// Mitsubishi GX Works2 project: STEP_SEQUENCE   PLC: Q02/Q02H

PROGRAM MAIN
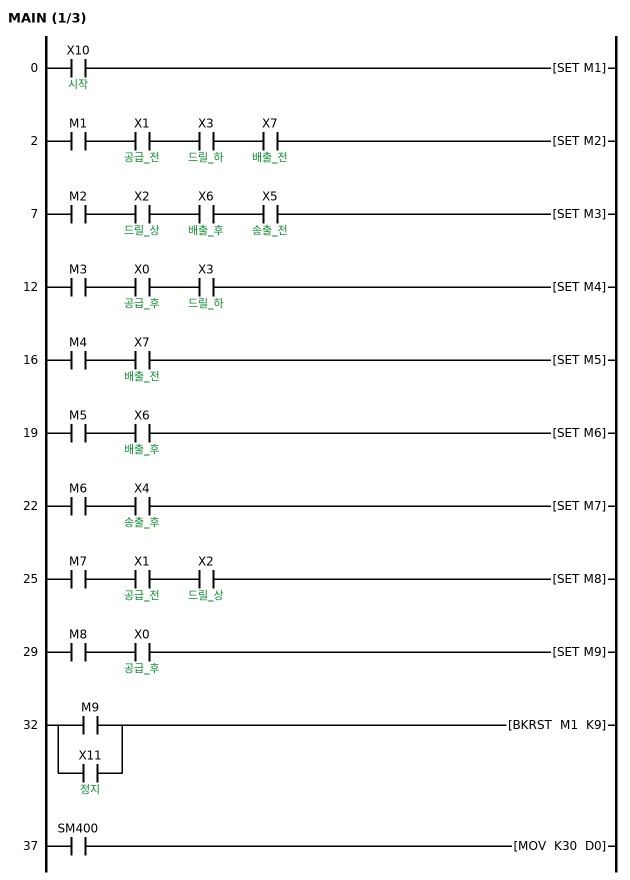
0     LD      X10  ; 시작
      SET     M1
2     LD      M1
      AND     X1  ; 공급_전
      AND     X3  ; 드릴_하
      AND     X7  ; 배출_전
      SET     M2
7     LD      M2
      AND     X2  ; 드릴_상
      AND     X6  ; 배출_후
      AND     X5  ; 송출_전
      SET     M3
12    LD      M3
      AND     X0  ; 공급_후
      AND     X3  ; 드릴_하
      SET     M4
16    LD      M4
      AND     X7  ; 배출_전
      SET     M5
19    LD      M5
      AND     X6  ; 배출_후
      SET     M6
22    LD      M6
      AND     X4  ; 송출_후
      SET     M7
25    LD      M7
      AND     X1  ; 공급_전
      AND     X2  ; 드릴_상
      SET     M8
29    LD      M8
      AND     X0  ; 공급_후
      SET     M9
32    LD      M9
      OR      X11  ; 정지
      BKRST   M1 K9
37    LD      SM400
      MOV     K30 D0
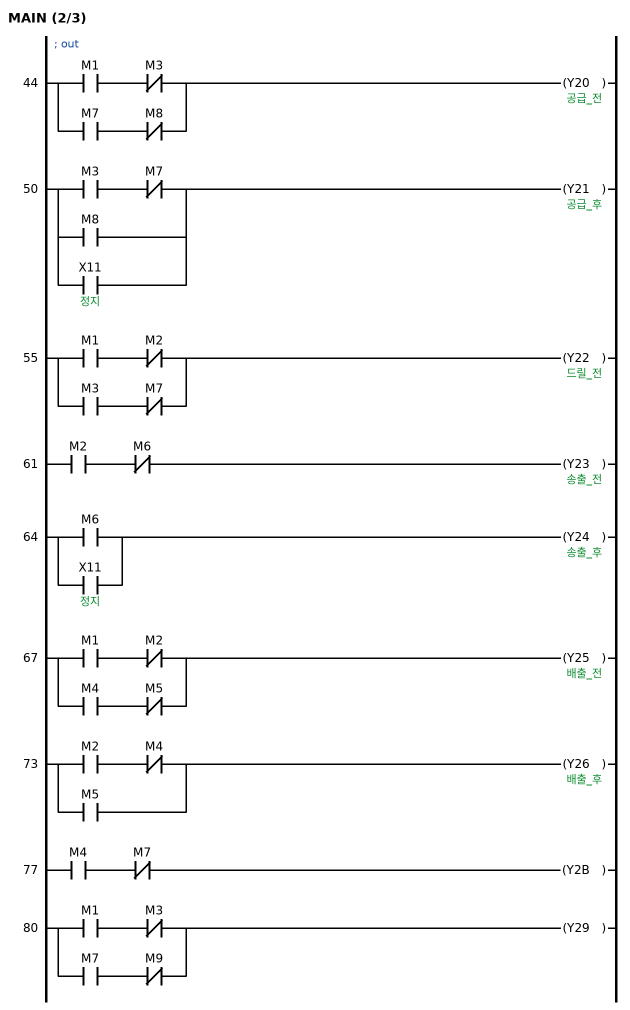
; out
44    LD      M1
      ANI     M3
      LD      M7
      ANI     M8
      ORB
      OUT     Y20  ; 공급_전
50    LD      M3
      ANI     M7
      OR      M8
      OR      X11  ; 정지
      OUT     Y21  ; 공급_후
55    LD      M1
      ANI     M2
      LD      M3
      ANI     M7
      ORB
      OUT     Y22  ; 드릴_전
61    LD      M2
      ANI     M6
      OUT     Y23  ; 송출_전
64    LD      M6
      OR      X11  ; 정지
      OUT     Y24  ; 송출_후
67    LD      M1
      ANI     M2
      LD      M4
      ANI     M5
      ORB
      OUT     Y25  ; 배출_전
73    LD      M2
      ANI     M4
      OR      M5
      OUT     Y26  ; 배출_후
77    LD      M4
      ANI     M7
      OUT     Y2B
80    LD      M1
      ANI     M3
      LD      M7
      ANI     M9
      ORB
      OUT     Y29
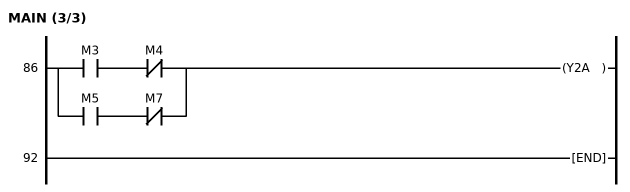
86    LD      M3
      ANI     M4
      LD      M5
      ANI     M7
      ORB
      OUT     Y2A
92    END
END_PROGRAM

PROGRAM APP1
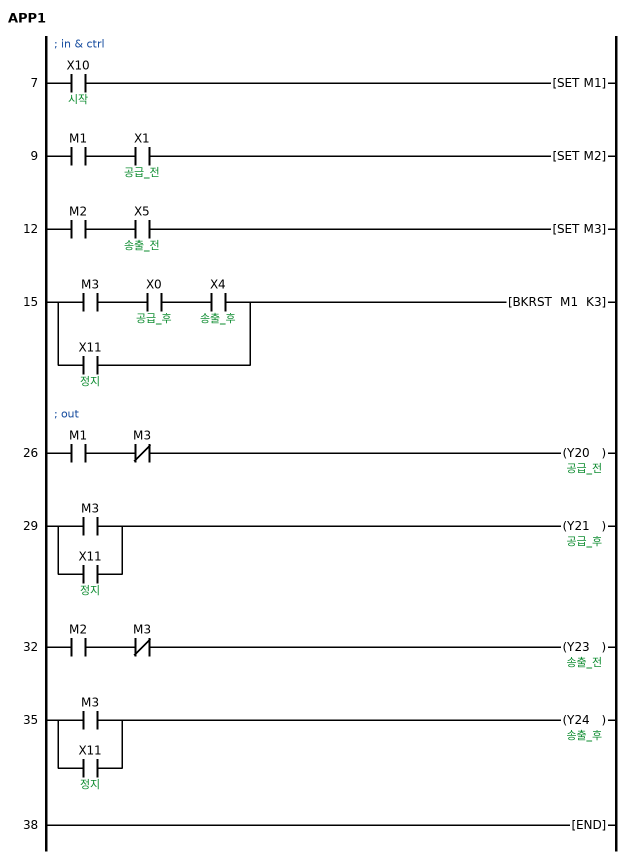
; in & ctrl
7     LD      X10  ; 시작
      SET     M1
9     LD      M1
      AND     X1  ; 공급_전
      SET     M2
12    LD      M2
      AND     X5  ; 송출_전
      SET     M3
15    LD      M3
      AND     X0  ; 공급_후
      AND     X4  ; 송출_후
      OR      X11  ; 정지
      BKRST   M1 K3
; out
26    LD      M1
      ANI     M3
      OUT     Y20  ; 공급_전
29    LD      M3
      OR      X11  ; 정지
      OUT     Y21  ; 공급_후
32    LD      M2
      ANI     M3
      OUT     Y23  ; 송출_전
35    LD      M3
      OR      X11  ; 정지
      OUT     Y24  ; 송출_후
38    END
END_PROGRAM

PROGRAM APP2
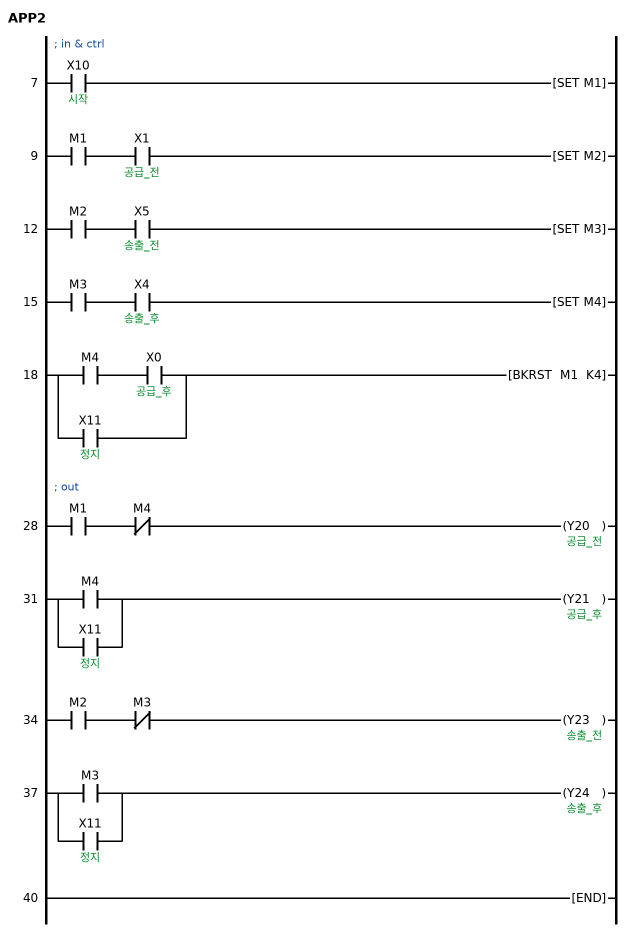
; in & ctrl
7     LD      X10  ; 시작
      SET     M1
9     LD      M1
      AND     X1  ; 공급_전
      SET     M2
12    LD      M2
      AND     X5  ; 송출_전
      SET     M3
15    LD      M3
      AND     X4  ; 송출_후
      SET     M4
18    LD      M4
      AND     X0  ; 공급_후
      OR      X11  ; 정지
      BKRST   M1 K4
; out
28    LD      M1
      ANI     M4
      OUT     Y20  ; 공급_전
31    LD      M4
      OR      X11  ; 정지
      OUT     Y21  ; 공급_후
34    LD      M2
      ANI     M3
      OUT     Y23  ; 송출_전
37    LD      M3
      OR      X11  ; 정지
      OUT     Y24  ; 송출_후
40    END
END_PROGRAM

PROGRAM APP3
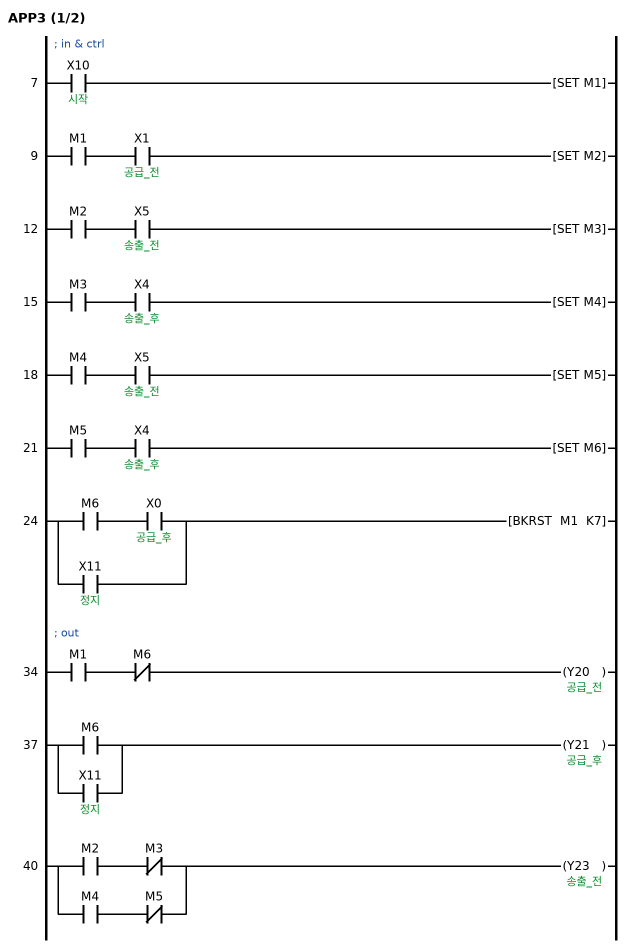
; in & ctrl
7     LD      X10  ; 시작
      SET     M1
9     LD      M1
      AND     X1  ; 공급_전
      SET     M2
12    LD      M2
      AND     X5  ; 송출_전
      SET     M3
15    LD      M3
      AND     X4  ; 송출_후
      SET     M4
18    LD      M4
      AND     X5  ; 송출_전
      SET     M5
21    LD      M5
      AND     X4  ; 송출_후
      SET     M6
24    LD      M6
      AND     X0  ; 공급_후
      OR      X11  ; 정지
      BKRST   M1 K7
; out
34    LD      M1
      ANI     M6
      OUT     Y20  ; 공급_전
37    LD      M6
      OR      X11  ; 정지
      OUT     Y21  ; 공급_후
40    LD      M2
      ANI     M3
      LD      M4
      ANI     M5
      ORB
      OUT     Y23  ; 송출_전
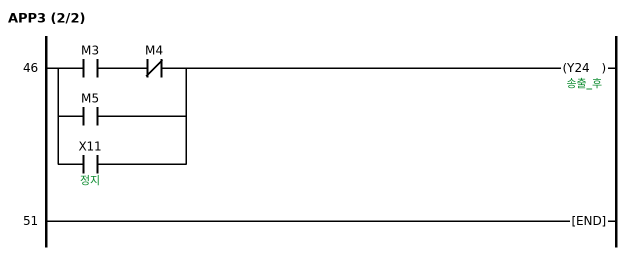
46    LD      M3
      ANI     M4
      OR      M5
      OR      X11  ; 정지
      OUT     Y24  ; 송출_후
51    END
END_PROGRAM

PROGRAM stepDoc
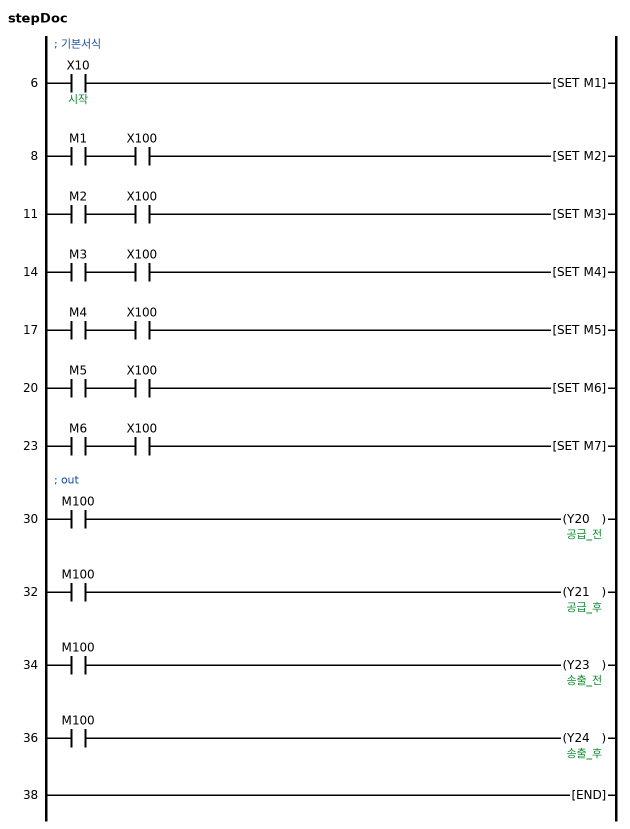
; 기본서식
6     LD      X10  ; 시작
      SET     M1
8     LD      M1
      AND     X100
      SET     M2
11    LD      M2
      AND     X100
      SET     M3
14    LD      M3
      AND     X100
      SET     M4
17    LD      M4
      AND     X100
      SET     M5
20    LD      M5
      AND     X100
      SET     M6
23    LD      M6
      AND     X100
      SET     M7
; out
30    LD      M100
      OUT     Y20  ; 공급_전
32    LD      M100
      OUT     Y21  ; 공급_후
34    LD      M100
      OUT     Y23  ; 송출_전
36    LD      M100
      OUT     Y24  ; 송출_후
38    END
END_PROGRAM

PROGRAM APP4
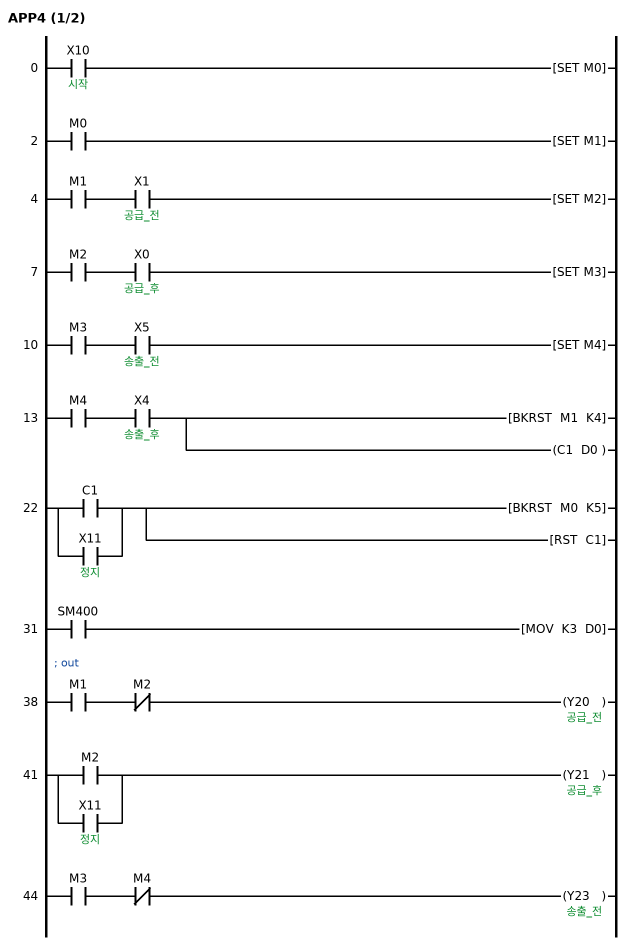
0     LD      X10  ; 시작
      SET     M0
2     LD      M0
      SET     M1
4     LD      M1
      AND     X1  ; 공급_전
      SET     M2
7     LD      M2
      AND     X0  ; 공급_후
      SET     M3
10    LD      M3
      AND     X5  ; 송출_전
      SET     M4
13    LD      M4
      AND     X4  ; 송출_후
      BKRST   M1 K4
      OUT     C1 D0
22    LD      C1
      OR      X11  ; 정지
      BKRST   M0 K5
      RST     C1
31    LD      SM400
      MOV     K3 D0
; out
38    LD      M1
      ANI     M2
      OUT     Y20  ; 공급_전
41    LD      M2
      OR      X11  ; 정지
      OUT     Y21  ; 공급_후
44    LD      M3
      ANI     M4
      OUT     Y23  ; 송출_전
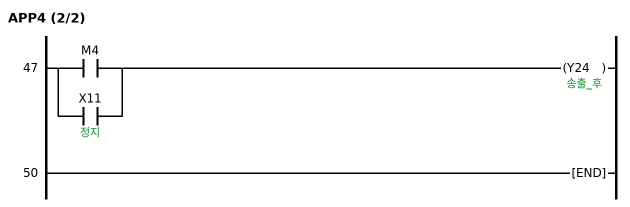
47    LD      M4
      OR      X11  ; 정지
      OUT     Y24  ; 송출_후
50    END
END_PROGRAM

PROGRAM APP3-1
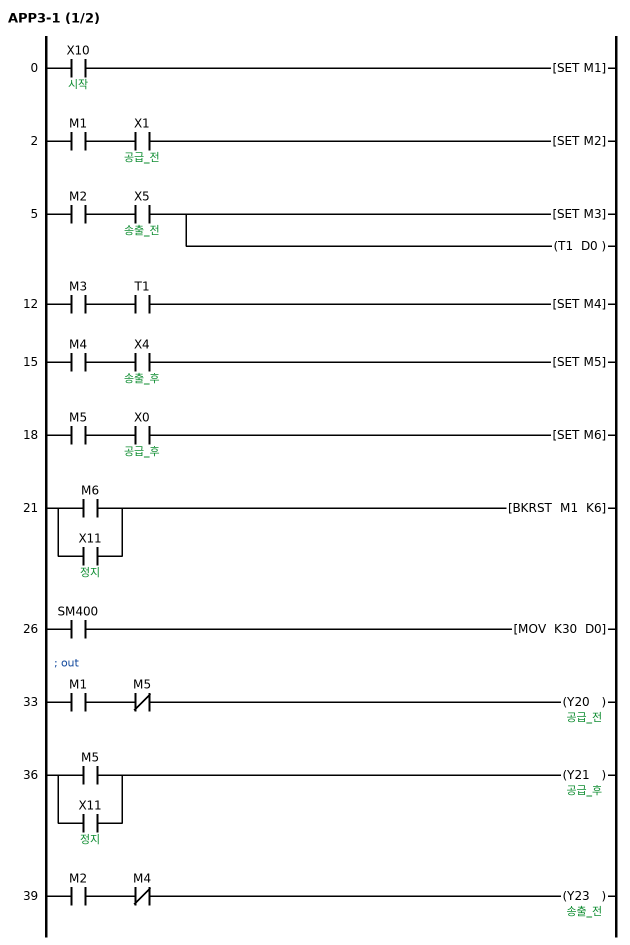
0     LD      X10  ; 시작
      SET     M1
2     LD      M1
      AND     X1  ; 공급_전
      SET     M2
5     LD      M2
      AND     X5  ; 송출_전
      SET     M3
      OUT     T1 D0
12    LD      M3
      AND     T1
      SET     M4
15    LD      M4
      AND     X4  ; 송출_후
      SET     M5
18    LD      M5
      AND     X0  ; 공급_후
      SET     M6
21    LD      M6
      OR      X11  ; 정지
      BKRST   M1 K6
26    LD      SM400
      MOV     K30 D0
; out
33    LD      M1
      ANI     M5
      OUT     Y20  ; 공급_전
36    LD      M5
      OR      X11  ; 정지
      OUT     Y21  ; 공급_후
39    LD      M2
      ANI     M4
      OUT     Y23  ; 송출_전
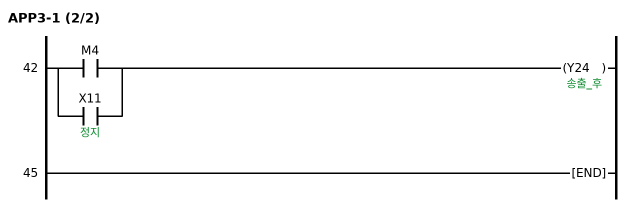
42    LD      M4
      OR      X11  ; 정지
      OUT     Y24  ; 송출_후
45    END
END_PROGRAM

PROGRAM complex1
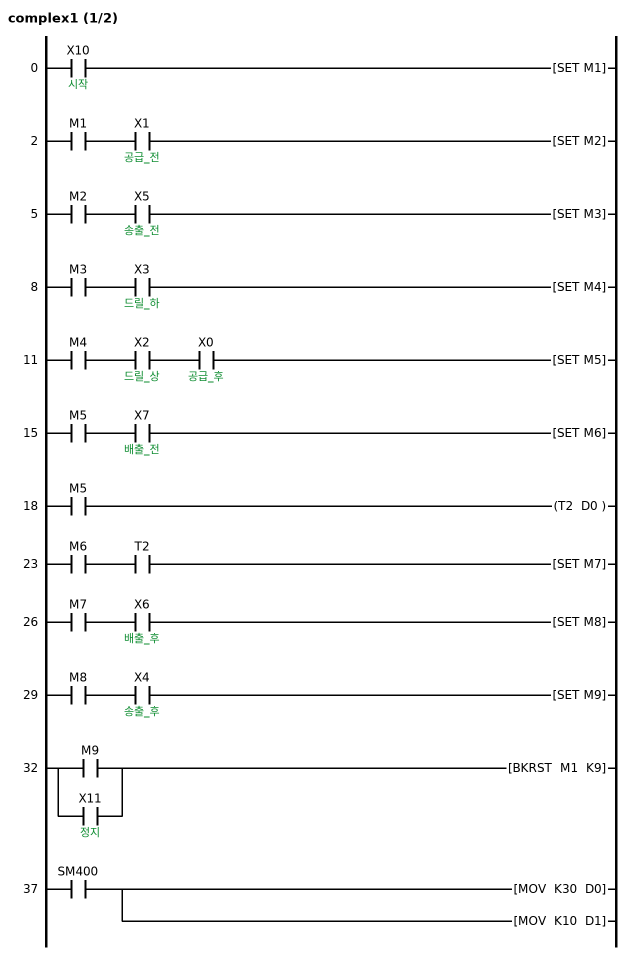
0     LD      X10  ; 시작
      SET     M1
2     LD      M1
      AND     X1  ; 공급_전
      SET     M2
5     LD      M2
      AND     X5  ; 송출_전
      SET     M3
8     LD      M3
      AND     X3  ; 드릴_하
      SET     M4
11    LD      M4
      AND     X2  ; 드릴_상
      AND     X0  ; 공급_후
      SET     M5
15    LD      M5
      AND     X7  ; 배출_전
      SET     M6
18    LD      M5
      OUT     T2 D0
23    LD      M6
      AND     T2
      SET     M7
26    LD      M7
      AND     X6  ; 배출_후
      SET     M8
29    LD      M8
      AND     X4  ; 송출_후
      SET     M9
32    LD      M9
      OR      X11  ; 정지
      BKRST   M1 K9
37    LD      SM400
      MOV     K30 D0
      MOV     K10 D1
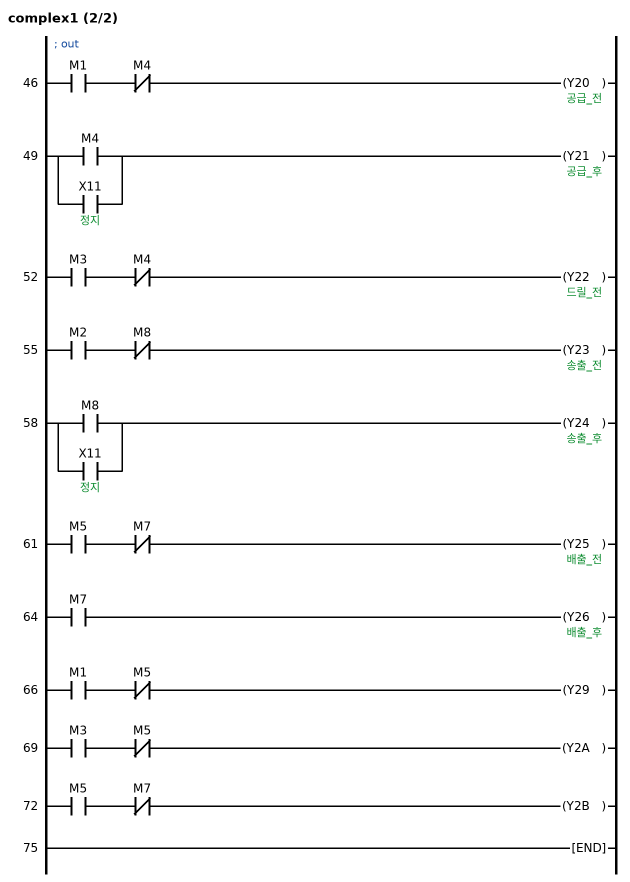
; out
46    LD      M1
      ANI     M4
      OUT     Y20  ; 공급_전
49    LD      M4
      OR      X11  ; 정지
      OUT     Y21  ; 공급_후
52    LD      M3
      ANI     M4
      OUT     Y22  ; 드릴_전
55    LD      M2
      ANI     M8
      OUT     Y23  ; 송출_전
58    LD      M8
      OR      X11  ; 정지
      OUT     Y24  ; 송출_후
61    LD      M5
      ANI     M7
      OUT     Y25  ; 배출_전
64    LD      M7
      OUT     Y26  ; 배출_후
66    LD      M1
      ANI     M5
      OUT     Y29
69    LD      M3
      ANI     M5
      OUT     Y2A
72    LD      M5
      ANI     M7
      OUT     Y2B
75    END
END_PROGRAM

PROGRAM complex2
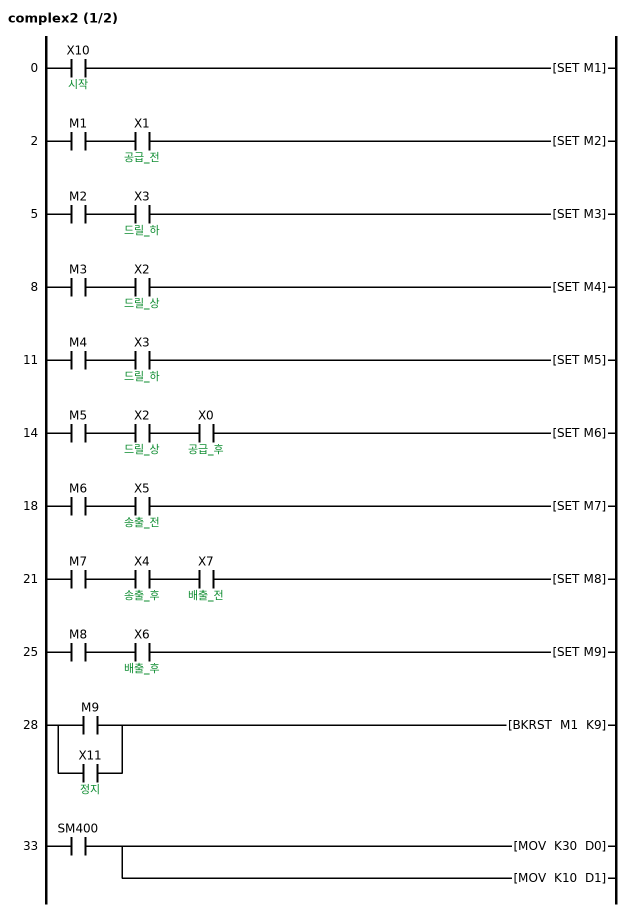
0     LD      X10  ; 시작
      SET     M1
2     LD      M1
      AND     X1  ; 공급_전
      SET     M2
5     LD      M2
      AND     X3  ; 드릴_하
      SET     M3
8     LD      M3
      AND     X2  ; 드릴_상
      SET     M4
11    LD      M4
      AND     X3  ; 드릴_하
      SET     M5
14    LD      M5
      AND     X2  ; 드릴_상
      AND     X0  ; 공급_후
      SET     M6
18    LD      M6
      AND     X5  ; 송출_전
      SET     M7
21    LD      M7
      AND     X4  ; 송출_후
      AND     X7  ; 배출_전
      SET     M8
25    LD      M8
      AND     X6  ; 배출_후
      SET     M9
28    LD      M9
      OR      X11  ; 정지
      BKRST   M1 K9
33    LD      SM400
      MOV     K30 D0
      MOV     K10 D1
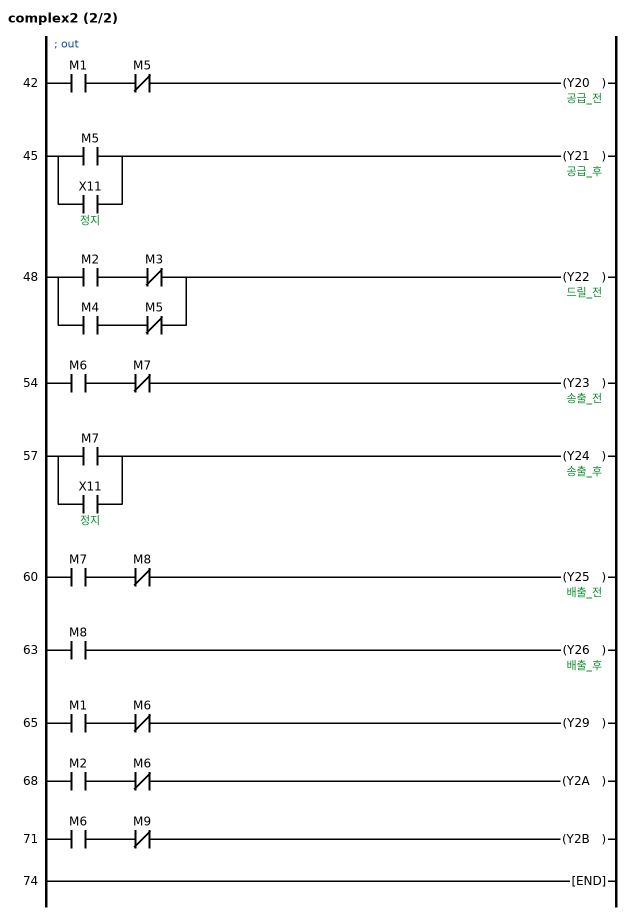
; out
42    LD      M1
      ANI     M5
      OUT     Y20  ; 공급_전
45    LD      M5
      OR      X11  ; 정지
      OUT     Y21  ; 공급_후
48    LD      M2
      ANI     M3
      LD      M4
      ANI     M5
      ORB
      OUT     Y22  ; 드릴_전
54    LD      M6
      ANI     M7
      OUT     Y23  ; 송출_전
57    LD      M7
      OR      X11  ; 정지
      OUT     Y24  ; 송출_후
60    LD      M7
      ANI     M8
      OUT     Y25  ; 배출_전
63    LD      M8
      OUT     Y26  ; 배출_후
65    LD      M1
      ANI     M6
      OUT     Y29
68    LD      M2
      ANI     M6
      OUT     Y2A
71    LD      M6
      ANI     M9
      OUT     Y2B
74    END
END_PROGRAM

PROGRAM complex3
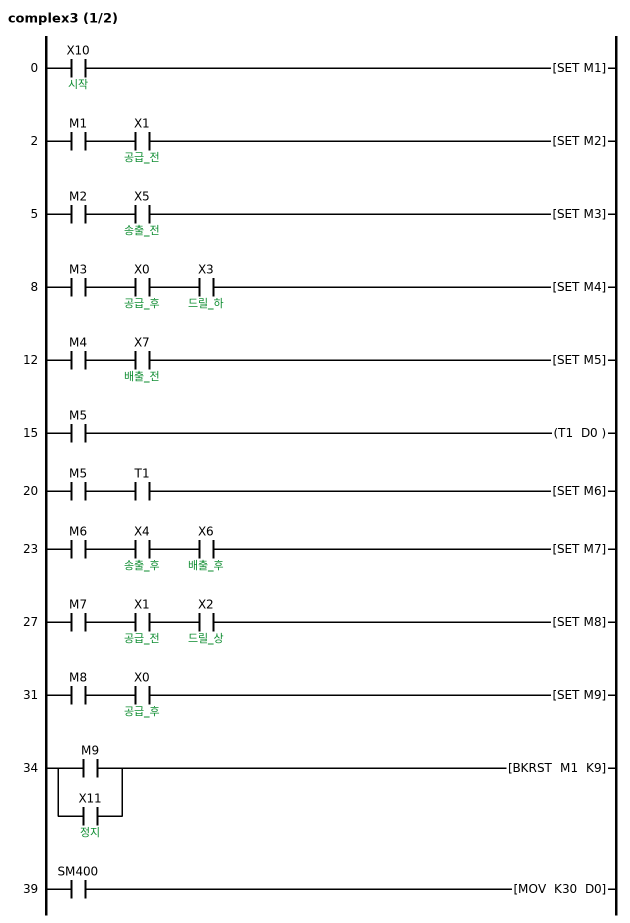
0     LD      X10  ; 시작
      SET     M1
2     LD      M1
      AND     X1  ; 공급_전
      SET     M2
5     LD      M2
      AND     X5  ; 송출_전
      SET     M3
8     LD      M3
      AND     X0  ; 공급_후
      AND     X3  ; 드릴_하
      SET     M4
12    LD      M4
      AND     X7  ; 배출_전
      SET     M5
15    LD      M5
      OUT     T1 D0
20    LD      M5
      AND     T1
      SET     M6
23    LD      M6
      AND     X4  ; 송출_후
      AND     X6  ; 배출_후
      SET     M7
27    LD      M7
      AND     X1  ; 공급_전
      AND     X2  ; 드릴_상
      SET     M8
31    LD      M8
      AND     X0  ; 공급_후
      SET     M9
34    LD      M9
      OR      X11  ; 정지
      BKRST   M1 K9
39    LD      SM400
      MOV     K30 D0
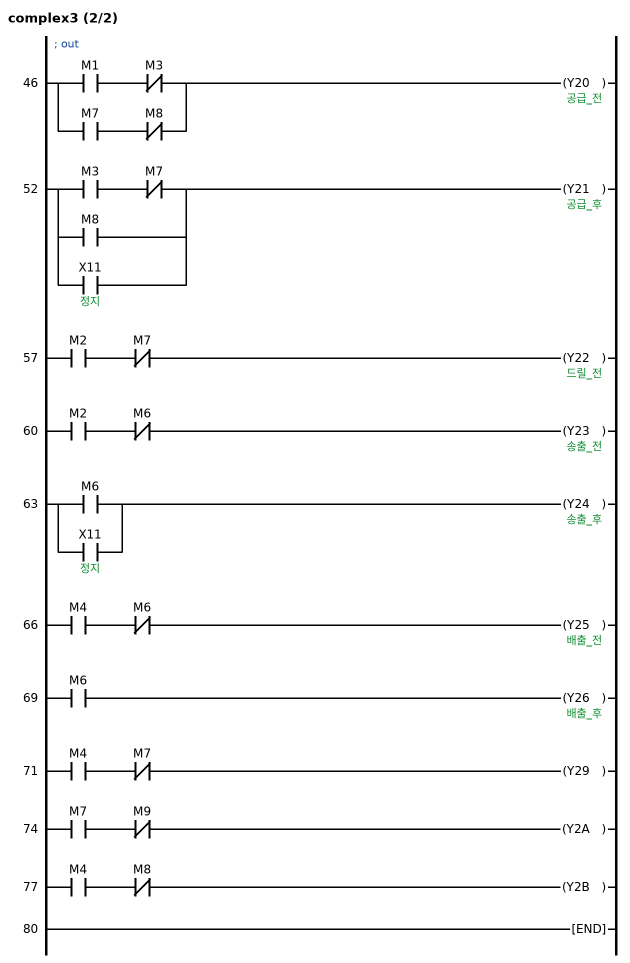
; out
46    LD      M1
      ANI     M3
      LD      M7
      ANI     M8
      ORB
      OUT     Y20  ; 공급_전
52    LD      M3
      ANI     M7
      OR      M8
      OR      X11  ; 정지
      OUT     Y21  ; 공급_후
57    LD      M2
      ANI     M7
      OUT     Y22  ; 드릴_전
60    LD      M2
      ANI     M6
      OUT     Y23  ; 송출_전
63    LD      M6
      OR      X11  ; 정지
      OUT     Y24  ; 송출_후
66    LD      M4
      ANI     M6
      OUT     Y25  ; 배출_전
69    LD      M6
      OUT     Y26  ; 배출_후
71    LD      M4
      ANI     M7
      OUT     Y29
74    LD      M7
      ANI     M9
      OUT     Y2A
77    LD      M4
      ANI     M8
      OUT     Y2B
80    END
END_PROGRAM

PROGRAM complex4
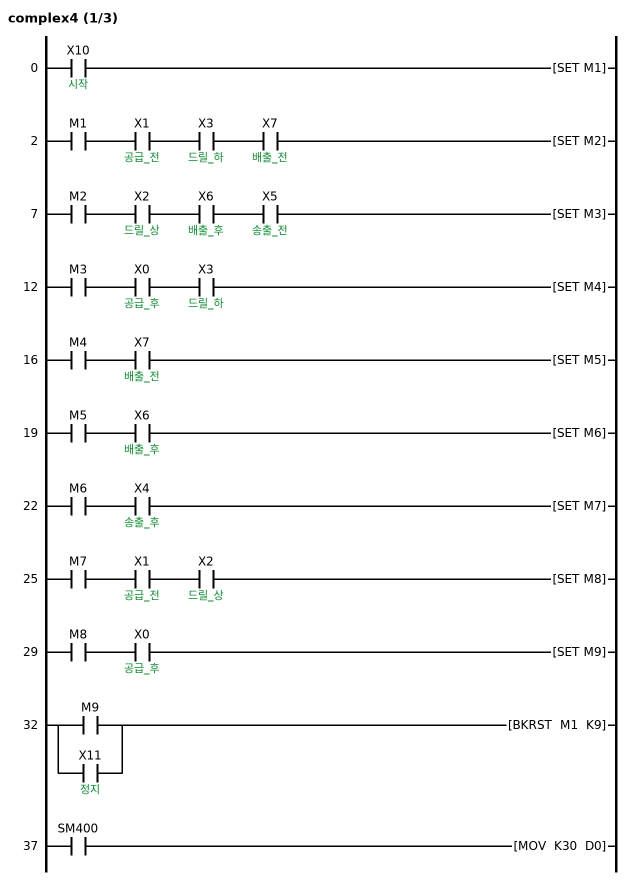
0     LD      X10  ; 시작
      SET     M1
2     LD      M1
      AND     X1  ; 공급_전
      AND     X3  ; 드릴_하
      AND     X7  ; 배출_전
      SET     M2
7     LD      M2
      AND     X2  ; 드릴_상
      AND     X6  ; 배출_후
      AND     X5  ; 송출_전
      SET     M3
12    LD      M3
      AND     X0  ; 공급_후
      AND     X3  ; 드릴_하
      SET     M4
16    LD      M4
      AND     X7  ; 배출_전
      SET     M5
19    LD      M5
      AND     X6  ; 배출_후
      SET     M6
22    LD      M6
      AND     X4  ; 송출_후
      SET     M7
25    LD      M7
      AND     X1  ; 공급_전
      AND     X2  ; 드릴_상
      SET     M8
29    LD      M8
      AND     X0  ; 공급_후
      SET     M9
32    LD      M9
      OR      X11  ; 정지
      BKRST   M1 K9
37    LD      SM400
      MOV     K30 D0
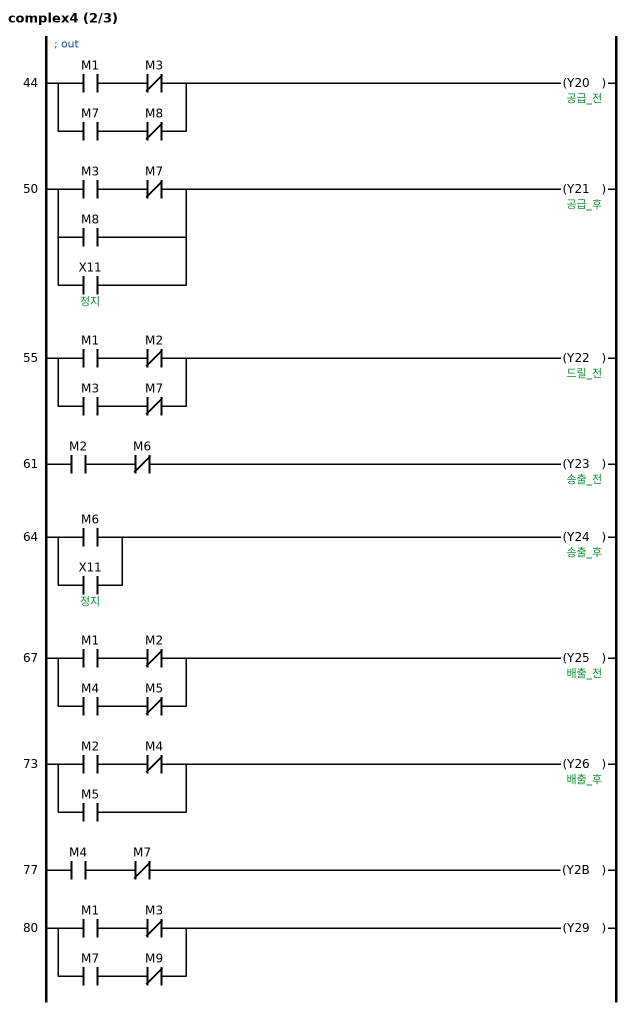
; out
44    LD      M1
      ANI     M3
      LD      M7
      ANI     M8
      ORB
      OUT     Y20  ; 공급_전
50    LD      M3
      ANI     M7
      OR      M8
      OR      X11  ; 정지
      OUT     Y21  ; 공급_후
55    LD      M1
      ANI     M2
      LD      M3
      ANI     M7
      ORB
      OUT     Y22  ; 드릴_전
61    LD      M2
      ANI     M6
      OUT     Y23  ; 송출_전
64    LD      M6
      OR      X11  ; 정지
      OUT     Y24  ; 송출_후
67    LD      M1
      ANI     M2
      LD      M4
      ANI     M5
      ORB
      OUT     Y25  ; 배출_전
73    LD      M2
      ANI     M4
      OR      M5
      OUT     Y26  ; 배출_후
77    LD      M4
      ANI     M7
      OUT     Y2B
80    LD      M1
      ANI     M3
      LD      M7
      ANI     M9
      ORB
      OUT     Y29
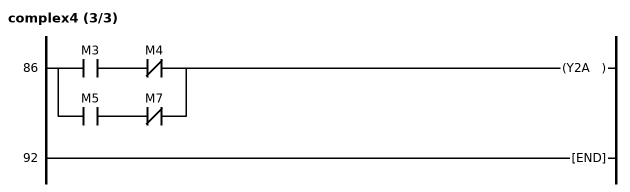
86    LD      M3
      ANI     M4
      LD      M5
      ANI     M7
      ORB
      OUT     Y2A
92    END
END_PROGRAM
